PROGRAM MAIN
VAR
END_VAR

END_PROGRAM

(* stored: Version 1.1.0.1
   POU MAIN: Id {7133b59b-9ac1-41be-8dde-d4c9b6401afa} *)
